LIN {X 0,Y 162.049,Z 553.984,A -85,B 0,C 180,E1 -30421.833,E2 -30421.833} C_VEL
LIN {X 0,Y 146.081,Z 553.984,A -85,B 0,C 180,E1 -30420.752,E2 -30420.752} C_VEL
LIN {X 0,Y 144.118,Z 551.984,A -85,B 0,C 180,E1 -30420.602,E2 -30420.602} C_VEL
LIN {X 0,Y 144.118,Z 543.325,A -85,B 0,C 180,E1 -30420.602,E2 -30420.602} C_VEL
LIN {X 0,Y 140.579,Z 542.113,A -85,B 0,C 180,E1 -30420.848,E2 -30420.848} C_VEL
LIN {X 0,Y 130.976,Z 554.064,A -85,B 0,C 180,E1 -30421.558,E2 -30421.558} C_VEL
LIN {X 0,Y 121.341,Z 564.22,A -85,B 0,C 180,E1 -30422.373,E2 -30422.373} C_VEL
LIN {X 0,Y 110.568,Z 573.82,A -85,B 0,C 180,E1 -30423.467,E2 -30423.467} C_VEL
LIN {X 0,Y 98.793,Z 582.692,A -85,B 0,C 180,E1 -30425.14,E2 -30425.14} C_VEL
LIN {X 0,Y 88.45,Z 589.309,A -85,B 0,C 180,E1 -30426.655,E2 -30426.655} C_VEL
LIN {X 0,Y 74.815,Z 596.611,A -85,B 0,C 180,E1 -30429.46,E2 -30429.46} C_VEL
LIN {X 0,Y 62.614,Z 601.95,A -85,B 0,C 180,E1 -30432.974,E2 -30432.974} C_VEL
LIN {X 0,Y 51.655,Z 605.807,A -85,B 0,C 180,E1 -30437.738,E2 -30437.738} C_VEL
LIN {X 0,Y 39.196,Z 609.257,A -85,B 0,C 180,E1 -30446.285,E2 -30446.285} C_VEL
LIN {X 0,Y 28.369,Z 611.515,A -85,B 0,C 180,E1 -30461.984,E2 -30461.984} C_VEL
LIN {X 0,Y 21.295,Z 612.65,A -85,B 0,C 180,E1 -30490.719,E2 -30490.719} C_VEL
LIN {X 0,Y 20.38,Z 612.797,A -85,B 0,C 180,E1 -30509.991,E2 -30509.991} C_VEL
LIN {X 0,Y 24.114,Z 612.247,A -85,B 0,C 180,E1 -30545.644,E2 -30545.644} C_VEL
LIN {X 0,Y 33.472,Z 610.592,A -85,B 0,C 180,E1 -30567.117,E2 -30567.117} C_VEL
LIN {X 0,Y 45.288,Z 607.778,A -85,B 0,C 180,E1 -30578.598,E2 -30578.598} C_VEL
LIN {X 0,Y 58.09,Z 603.739,A -85,B 0,C 180,E1 -30585.427,E2 -30585.427} C_VEL
LIN {X 0,Y 71.412,Z 598.368,A -85,B 0,C 180,E1 -30589.771,E2 -30589.771} C_VEL
LIN {X 0,Y 85.005,Z 591.513,A -85,B 0,C 180,E1 -30592.792,E2 -30592.792} C_VEL
LIN {X 0,Y 97.044,Z 584.138,A -85,B 0,C 180,E1 -30594.719,E2 -30594.719} C_VEL
LIN {X 0,Y 109.136,Z 575.255,A -85,B 0,C 180,E1 -30596.459,E2 -30596.459} C_VEL
LIN {X 0,Y 119.584,Z 566.168,A -85,B 0,C 180,E1 -30597.529,E2 -30597.529} C_VEL
LIN {X 0,Y 130.063,Z 555.447,A -85,B 0,C 180,E1 -30598.44,E2 -30598.44} C_VEL
LIN {X 0,Y 139.694,Z 543.733,A -85,B 0,C 180,E1 -30599.159,E2 -30599.159} C_VEL
LIN {X 0,Y 140.57,Z 542.566,A -85,B 0,C 180,E1 -30599.226,E2 -30599.226} C_VEL
LIN {X 0,Y 140.564,Z 542.586,A -85,B 0,C 180,E1 -30599.446,E2 -30599.446} C_VEL
LIN {X 0,Y 131.162,Z 554.306,A -85,B 0,C 180,E1 -30600,E2 -30600} C_VEL
LIN {X 0,Y 121.24,Z 564.795,A -85,B 0,C 180,E1 -30600.741,E2 -30600.741} C_VEL
LIN {X 0,Y 108.979,Z 575.629,A -85,B 0,C 180,E1 -30601.701,E2 -30601.701} C_VEL
LIN {X 0,Y 96.766,Z 584.669,A -85,B 0,C 180,E1 -30603.014,E2 -30603.014} C_VEL
LIN {X 0,Y 84.636,Z 592.188,A -85,B 0,C 180,E1 -30604.85,E2 -30604.85} C_VEL
LIN {X 0,Y 70.921,Z 599.21,A -85,B 0,C 180,E1 -30607.73,E2 -30607.73} C_VEL
LIN {X 0,Y 57.45,Z 604.742,A -85,B 0,C 180,E1 -30611.872,E2 -30611.872} C_VEL
LIN {X 0,Y 44.474,Z 608.943,A -85,B 0,C 180,E1 -30618.544,E2 -30618.544} C_VEL
LIN {X 0,Y 32.512,Z 611.905,A -85,B 0,C 180,E1 -30630.168,E2 -30630.168} C_VEL
LIN {X 0,Y 23.144,Z 613.693,A -85,B 0,C 180,E1 -30652.613,E2 -30652.613} C_VEL
LIN {X 0,Y 20.022,Z 614.336,A -85,B 0,C 180,E1 -30690.01,E2 -30690.01} C_VEL
LIN {X 0,Y 23.148,Z 613.669,A -85,B 0,C 180,E1 -30727.401,E2 -30727.401} C_VEL
LIN {X 0,Y 32.52,Z 611.848,A -85,B 0,C 180,E1 -30749.831,E2 -30749.831} C_VEL
LIN {X 0,Y 44.822,Z 608.755,A -85,B 0,C 180,E1 -30761.725,E2 -30761.725} C_VEL
LIN {X 0,Y 57.453,Z 604.629,A -85,B 0,C 180,E1 -30768.147,E2 -30768.147} C_VEL
LIN {X 0,Y 70.925,Z 599.059,A -85,B 0,C 180,E1 -30772.286,E2 -30772.286} C_VEL
LIN {X 0,Y 84.986,Z 591.782,A -85,B 0,C 180,E1 -30775.257,E2 -30775.257} C_VEL
LIN {X 0,Y 98.515,Z 583.217,A -85,B 0,C 180,E1 -30777.184,E2 -30777.184} C_VEL
LIN {X 0,Y 110.734,Z 573.912,A -85,B 0,C 180,E1 -30778.479,E2 -30778.479} C_VEL
LIN {X 0,Y 121.246,Z 564.473,A -85,B 0,C 180,E1 -30779.274,E2 -30779.274} C_VEL
LIN {X 0,Y 131.998,Z 553.003,A -85,B 0,C 180,E1 -30780.054,E2 -30780.054} C_VEL
LIN {X 0,Y 140.571,Z 542.139,A -85,B 0,C 180,E1 -30780.569,E2 -30780.569} C_VEL
LIN {X 0,Y 140.579,Z 542.113,A -85,B 0,C 180,E1 -30780.848,E2 -30780.848} C_VEL
LIN {X 0,Y 140.625,Z 544.112,A -85,B 0,C 180,E1 -30781.694,E2 -30781.694} C_VEL
LIN {X 0,Y 140.625,Z 597.415,A -85,B 0,C 180,E1 -30781.694,E2 -30781.694} C_VEL
LIN {X 0,Y 96.397,Z 597.415,A -85,B 0,C 180,E1 -30781.32,E2 -30781.32} C_VEL
LIN {X 0,Y 94.398,Z 595.415,A -85,B 0,C 180,E1 -30781.295,E2 -30781.295} C_VEL
LIN {X 0,Y 94.398,Z 589.214,A -85,B 0,C 180,E1 -30781.295,E2 -30781.295} C_VEL
LIN {X 0,Y 91.404,Z 587.505,A -85,B 0,C 180,E1 -30781.618,E2 -30781.618} C_VEL
LIN {X 0,Y 77.452,Z 595.225,A -85,B 0,C 180,E1 -30783.454,E2 -30783.454} C_VEL
LIN {X 0,Y 63.602,Z 601.359,A -85,B 0,C 180,E1 -30785.981,E2 -30785.981} C_VEL
LIN {X 0,Y 49.945,Z 606.079,A -85,B 0,C 180,E1 -30789.914,E2 -30789.914} C_VEL
LIN {X 0,Y 36.602,Z 609.529,A -85,B 0,C 180,E1 -30796.229,E2 -30796.229} C_VEL
LIN {X 0,Y 24.186,Z 611.787,A -85,B 0,C 180,E1 -30809.323,E2 -30809.323} C_VEL
LIN {X 0,Y 14.773,Z 612.921,A -85,B 0,C 180,E1 -30841.577,E2 -30841.577} C_VEL
LIN {X 0,Y 13.3,Z 613.066,A -85,B 0,C 180,E1 -30869.985,E2 -30869.985} C_VEL
LIN {X 0,Y 18.802,Z 612.518,A -85,B 0,C 180,E1 -30918.366,E2 -30918.366} C_VEL
LIN {X 0,Y 30.205,Z 610.863,A -85,B 0,C 180,E1 -30938.526,E2 -30938.526} C_VEL
LIN {X 0,Y 43.197,Z 608.049,A -85,B 0,C 180,E1 -30947.45,E2 -30947.45} C_VEL
LIN {X 0,Y 56.718,Z 604.009,A -85,B 0,C 180,E1 -30952.405,E2 -30952.405} C_VEL
LIN {X 0,Y 70.496,Z 598.638,A -85,B 0,C 180,E1 -30955.485,E2 -30955.485} C_VEL
LIN {X 0,Y 84.407,Z 591.783,A -85,B 0,C 180,E1 -30957.603,E2 -30957.603} C_VEL
LIN {X 0,Y 91.394,Z 587.732,A -85,B 0,C 180,E1 -30958.452,E2 -30958.452} C_VEL
LIN {X 0,Y 91.369,Z 587.778,A -85,B 0,C 180,E1 -30959.217,E2 -30959.217} C_VEL
LIN {X 0,Y 77.314,Z 595.626,A -85,B 0,C 180,E1 -30960.878,E2 -30960.878} C_VEL
LIN {X 0,Y 63.344,Z 601.877,A -85,B 0,C 180,E1 -30963.136,E2 -30963.136} C_VEL
LIN {X 0,Y 49.533,Z 606.729,A -85,B 0,C 180,E1 -30966.721,E2 -30966.721} C_VEL
LIN {X 0,Y 36.054,Z 610.301,A -85,B 0,C 180,E1 -30972.954,E2 -30972.954} C_VEL
LIN {X 0,Y 23.409,Z 612.668,A -85,B 0,C 180,E1 -30985.771,E2 -30985.771} C_VEL
LIN {X 0,Y 14.048,Z 613.888,A -85,B 0,C 180,E1 -31019.997,E2 -31019.997} C_VEL
LIN {X 0,Y 12.913,Z 614.065,A -85,B 0,C 180,E1 -31050.015,E2 -31050.015} C_VEL
LIN {X 0,Y 17.996,Z 613.396,A -85,B 0,C 180,E1 -31101.376,E2 -31101.376} C_VEL
LIN {X 0,Y 29.578,Z 611.575,A -85,B 0,C 180,E1 -31121.908,E2 -31121.908} C_VEL
LIN {X 0,Y 42.739,Z 608.583,A -85,B 0,C 180,E1 -31130.649,E2 -31130.649} C_VEL
LIN {X 0,Y 56.417,Z 604.355,A -85,B 0,C 180,E1 -31135.298,E2 -31135.298} C_VEL
LIN {X 0,Y 70.323,Z 598.784,A -85,B 0,C 180,E1 -31138.092,E2 -31138.092} C_VEL
LIN {X 0,Y 84.34,Z 591.713,A -85,B 0,C 180,E1 -31140.057,E2 -31140.057} C_VEL
LIN {X 0,Y 91.376,Z 587.556,A -85,B 0,C 180,E1 -31140.784,E2 -31140.784} C_VEL
LIN {X 0,Y 91.404,Z 587.505,A -85,B 0,C 180,E1 -31141.618,E2 -31141.618} C_VEL
LIN {X 0,Y 91.486,Z 589.504,A -85,B 0,C 180,E1 -31142.918,E2 -31142.918} C_VEL
LIN {X 0,Y 91.486,Z 616.065,A -85,B 0,C 180,E1 -31142.918,E2 -31142.918} C_VEL
LIN {X 0,Y 53.7,Z 616.065,A -85,B 0,C 180,E1 -31141.407,E2 -31141.407} C_VEL
LIN {X 0,Y 51.704,Z 614.065,A -85,B 0,C 180,E1 -31141.266,E2 -31141.266} C_VEL
LIN {X 0,Y 51.704,Z 608.286,A -85,B 0,C 180,E1 -31141.266,E2 -31141.266} C_VEL
LIN {X 0,Y 49.221,Z 606.352,A -85,B 0,C 180,E1 -31141.695,E2 -31141.695} C_VEL
LIN {X 0,Y 35.28,Z 609.801,A -85,B 0,C 180,E1 -31145.046,E2 -31145.046} C_VEL
LIN {X 0,Y 21.61,Z 612.058,A -85,B 0,C 180,E1 -31152.627,E2 -31152.627} C_VEL
LIN {X 0,Y 9.178,Z 613.191,A -85,B 0,C 180,E1 -31179.992,E2 -31179.992} C_VEL
LIN {X 0,Y 6.203,Z 613.337,A -85,B 0,C 180,E1 -31229.969,E2 -31229.969} C_VEL
LIN {X 0,Y 15.044,Z 612.789,A -85,B 0,C 180,E1 -31299.087,E2 -31299.087} C_VEL
LIN {X 0,Y 28.382,Z 611.134,A -85,B 0,C 180,E1 -31312.047,E2 -31312.047} C_VEL
LIN {X 0,Y 42.225,Z 608.32,A -85,B 0,C 180,E1 -31316.945,E2 -31316.945} C_VEL
LIN {X 0,Y 48.336,Z 606.727,A -85,B 0,C 180,E1 -31318.524,E2 -31318.524} C_VEL
LIN {X 0,Y 35.148,Z 610.028,A -85,B 0,C 180,E1 -31321.465,E2 -31321.465} C_VEL
LIN {X 0,Y 21.296,Z 612.396,A -85,B 0,C 180,E1 -31328.146,E2 -31328.146} C_VEL
LIN {X 0,Y 8.635,Z 613.616,A -85,B 0,C 180,E1 -31355.562,E2 -31355.562} C_VEL
LIN {X 0,Y 5.792,Z 613.794,A -85,B 0,C 180,E1 -31410.033,E2 -31410.033} C_VEL
LIN {X 0,Y 14.635,Z 613.123,A -85,B 0,C 180,E1 -31483.872,E2 -31483.872} C_VEL
LIN {X 0,Y 28.186,Z 611.3,A -85,B 0,C 180,E1 -31495.932,E2 -31495.932} C_VEL
LIN {X 0,Y 42.172,Z 608.308,A -85,B 0,C 180,E1 -31500.326,E2 -31500.326} C_VEL
LIN {X 0,Y 49.221,Z 606.352,A -85,B 0,C 180,E1 -31501.695,E2 -31501.695} C_VEL
LIN {X 0,Y 49.221,Z 606.352,A -85,B 0,C 180,E1 -31501.695,E2 -31501.695}

QRS_NEXT_CUT()

QRS_NEXT()
QRS_HOME()

END
